// TIA Portal V18 export
VAR_GLOBAL   // PLC tag table "Default variable table"
   Clock_Byte AT %MB0 : Byte;
   System_Byte AT %MB1 : Byte;
   FirstScan AT %M1.0 : Bool;
   DiagStatusUpdate AT %M1.1 : Bool;
   AlwaysTRUE AT %M1.2 : Bool;
   AlwaysFALSE AT %M1.3 : Bool;
   "调试专用-DEBUG" AT %M12.1 : Bool;
   Tag_1 AT %M10.0 : Bool;   // 复位信号灯
   Tag_2 AT %M888.0 : Bool;
   Tag_3 AT %M100.1 : Bool;
   Tag_4 AT %M100.0 : Bool;
   Tag_77 AT %M200.0 : Bool;
   Tag_78 AT %M200.1 : Bool;
   Tag_79 AT %M200.2 : Bool;
   Tag_80 AT %MW100 : Int;
   Tag_81 AT %M30.0 : Bool;
   Tag_82 AT %MW102 : Int;
   Tag_83 AT %M200.3 : Bool;
   Tag_84 AT %M200.4 : Bool;
   Tag_93 AT %M200.5 : Bool;
   Tag_94 AT %M200.6 : Bool;
   Tag_95 AT %Q201.0 : Bool;
   Tag_96 AT %M201.0 : Bool;
   Tag_97 AT %M201.1 : Bool;
   Tag_98 AT %M100.2 : Bool;
   Tag_99 AT %M100.3 : Bool;
   Tag_100 AT %M100.4 : Bool;
   Tag_109 AT %M100.5 : Bool;
   Tag_110 AT %M100.6 : Bool;
   Tag_111 AT %M100.7 : Bool;
   Tag_112 AT %M101.0 : Bool;
   Tag_113 AT %M101.1 : Bool;
   Tag_114 AT %M101.2 : Bool;
   Tag_115 AT %M101.3 : Bool;
   Tag_116 AT %M101.4 : Bool;
   Tag_117 AT %M101.5 : Bool;
   Tag_118 AT %M101.6 : Bool;
   Tag_61 AT %M23.0 : Bool;
   Tag_62 AT %M23.1 : Bool;
   Tag_5 AT %M50.0 : Bool;
   Tag_6 AT %M50.1 : Bool;
   Tag_7 AT %M50.2 : Bool;
   Tag_8 AT %M60.0 : Bool;
   Tag_9 AT %M60.1 : Bool;
   Tag_10 AT %M300.0 : Bool;
   Tag_11 AT %M300.1 : Bool;
   Tag_12 AT %M300.2 : Bool;
   Tag_13 AT %M32.0 : Bool;
   Tag_14 AT %M36.0 : Bool;
   Tag_15 AT %M30.6 : Bool;
   Tag_16 AT %M55.0 : Bool;
   Tag_17 AT %M55.1 : Bool;
   Tag_18 AT %M62.3 : Bool;
   Tag_19 AT %M64.0 : Bool;
   Tag_20 AT %M666.6 : Bool;
   Tag_21 AT %M665.2 : Bool;
   Tag_22 AT %M56.3 : Bool;
   Tag_23 AT %M66.3 : Bool;
   Tag_24 AT %M323.0 : Bool;
   Tag_25 AT %M653.3 : Bool;
   Tag_26 AT %M456.0 : Bool;
   Tag_27 AT %M45.3 : Bool;
   Tag_28 AT %M45.4 : Bool;
   Tag_29 AT %M65.3 : Bool;
   Tag_30 AT %M55.5 : Bool;
   Tag_31 AT %M44.4 : Bool;
   Tag_32 AT %M55.6 : Bool;
   Tag_33 AT %M98.2 : Bool;
   Tag_34 AT %M98.6 : Bool;
   Tag_35 AT %M98.7 : Bool;
   Tag_36 AT %M96.3 : Bool;
END_VAR
